{attribute 'GeneratedUsingTerminal: AES-D-BC-ECAT-0000'}
{attribute addProperty BoxType "AES-D-BC-ECAT-0000"}
{attribute addProperty Id "digital_Data_OAT %Q*ARRAY[0..27] OF USINT28"}
{attribute addProperty CRC "3096397179"}
{attribute addProperty Size "28"}
TYPE Outputs_79BC345B EXTENDS TcoIo.OutputBase_10CEE7DE :
STRUCT
	{attribute addProperty Name "digital_Data_O"}
	digital_Data_O AT %Q* : ARRAY[0..27] OF USINT;
END_STRUCT
END_TYPE

(* stored: Version 1.2.0.0, ProductVersion 3.1.4024.11
   DUT Outputs_79BC345B: Id {4ac1196c-6f63-0d84-1877-d14f4bb1fc15} *)
